FUNCTION_BLOCK CU00xGround EXTENDS TcoTaskedSequencer
VAR
END_VAR

IF(Step(100, TRUE, 'FIRST STEP')) THEN
	StepCompleteWhen(TRUE);
END_IF

IF(Step(10000, TRUE, 'LAST STEP')) THEN
	_task.DoneWhen(TRUE);
END_IF

(*~
	<docu>
		<summary>
			Main method of the sequener. Custom code needs to be placed here. The sequencer is executed by call of **Instance.Run()** method.
			This method is abstract, and it must be overridden in derived block.
		</summary>
	</docu>
~*)
METHOD PROTECTED   Main : BOOL
END_METHOD

PROPERTY Station : REFERENCE TO CU00x
GET
VAR
    _station : POINTER TO CU00x;
END_VAR
IF __QUERYPOINTER(Parent,_station) THEN // Check if _Parent is Station001
	Station REF= _station^;              // If the check is successful dereference a pointer. simlar to THIS^ or SUPER^
END_IF
END_GET
END_PROPERTY

END_FUNCTION_BLOCK

(* stored: Version 1.1.0.1, ProductVersion 3.1.4024.9
   POU CU00xGround: Id {ea798b9b-c255-4bc1-bc0e-66e2dbced7d9}, SpecialFunc None
   Method Main: Id {0f44b6c1-dae2-4888-a3a0-6a44fd813a80}
   Property Station: Id {f5f158e7-8f54-483b-8ef9-070bf6fa1248}
   Get Get: Id {fecf57ba-7b86-4b09-b4c9-79cd0e6e6559} *)
